VAR
	_bComplete: BOOL; // True if the routing finishes
	_intRet: INT; // Return string converted to an integer
	_bResult : BOOL; // Output of the method
END_VAR
_bResult := FALSE;
bMGetLaserActivatedStatusBusy := TRUE;
_inst_intStep := intMGetLaserActivatedStatusStep;
CASE _inst_intStep OF
	0: // Wait for no error and router not busy
		IF NOT THIS^.P_bError AND NOT bRouterBusy THEN
			bRouterBusy := TRUE;
			_inst_intStep := _inst_intStep + 10;
		END_IF
		
	10: // Initialize parameters
		THIS^.M_LogMessage(_strSTART_MSG);
		_inst_fbParams.M_ClearParameters();
		// ADD ANY PARAMETERS HERE
		_inst_fbParams.M_OutputToParameterList(_inst_arrParams);
		_inst_intStep := _inst_intStep + 10;
		
	20: // Route the command
		_bComplete := M_RouterHelper(
			_in_strMethodName := _strCOMMAND_NAME, 
			_in_timeTimeout := _timeCOMMAND_TIMEOUT,
			_inout_arrParams := _inst_arrParams,
			_inout_arrOutputs := _inst_arrOutputs,
			_out_strReturnValue=>_inst_strRet);
		
		// If route completed, move to next step
		IF _bComplete THEN
			_inst_intStep := _inst_intStep + 10;
			bRouterBusy := FALSE;
		ELSIF THIS^.P_bError THEN
			_inst_intStep := 0;
			bRouterBusy := FALSE;
		END_IF
		
	30: // Parse results
		_intRet := STRING_TO_INT(_inst_strRet);
		IF _intRet > 0 THEN
			_bResult := TRUE;
			THIS^.M_LogMessage(_strEND_MSG);
			// DO ANY PARSING HERE
			_inst_fbParams.M_LoadFromParameterList(_inst_arrOutputs);
			out_IsLaserActivated := _inst_fbParams.M_ParseBool(_inst_fbParams.M_GetParameter('out_IsLaserActivated'));
			bConnected := TRUE;
		// Set error if command failed
		ELSE
			THIS^.M_SetError(_udintERROR_ID, _strERROR_MSG);
		END_IF
		// Go back to start
		_inst_intStep := 0;
END_CASE
M_GetLaserActivatedStatus := _bResult;
intMGetLaserActivatedStatusStep := _inst_intStep;
END_METHOD

METHOD PUBLIC M_GetLaserErrorStatus : BOOL
VAR_INPUT
//	LaserProgramFolderPath : STRING;
END_VAR
VAR_OUTPUT
	out_bool_IsLaserError : BOOL;
END_VAR
VAR CONSTANT
	_strCOMMAND_NAME : T_MaxString	:= 'GetLaserErrorStatus'; // Name of the API method
	_timeCOMMAND_TIMEOUT : TIME		:= T#30S; // Max time to receive API response
	_strSTART_MSG : T_MaxString		:= 'GettingLaserErrorStatus'; // Prints when method starts
	_strEND_MSG : T_MaxString		:= 'ReceivedLaserErrorStatus'; // Prints when method finishes
	_udintERROR_ID : UDINT			:= KeyenceLaserMarkerMDX2000_Error.FailedToGetLaserErrorStatus; // Error ID to set if command fails
	_strERROR_MSG : T_MaxString		:= 'Failed to Get Laser Error Status from Laser Marker!'; // Error message to set if command fails
END_VAR

VAR_INST
	_inst_arrParams: T_ApiParameterList; // Parameters array
	_inst_arrOutputs: T_ApiParameterList; // Outputs array
	_inst_strRet: T_ApiParamValue; // Return string from the router
	_inst_intStep: INT; // Current method step
	_inst_fbParams: FB_ApiParamBuilder; // Parameter builder FB
END_VAR

VAR
	_bComplete: BOOL; // True if the routing finishes
	_intRet: INT; // Return string converted to an integer
	_bResult : BOOL; // Output of the method
END_VAR
_bResult := FALSE;
bMGetLaserErrorStatusBusy := TRUE;
_inst_intStep := intMGetLaserErrorStatusStep;
CASE _inst_intStep OF
	0: // Wait for no error and router not busy
		IF NOT THIS^.P_bError AND NOT bRouterBusy THEN
			bRouterBusy := TRUE;
			_inst_intStep := _inst_intStep + 10;
		END_IF
		
	10: // Initialize parameters
		THIS^.M_LogMessage(_strSTART_MSG);
		_inst_fbParams.M_ClearParameters();
		// ADD ANY PARAMETERS HERE
		_inst_fbParams.M_OutputToParameterList(_inst_arrParams);
		_inst_intStep := _inst_intStep + 10;
		
	20: // Route the command
		_bComplete := M_RouterHelper(
			_in_strMethodName := _strCOMMAND_NAME, 
			_in_timeTimeout := _timeCOMMAND_TIMEOUT,
			_inout_arrParams := _inst_arrParams,
			_inout_arrOutputs := _inst_arrOutputs,
			_out_strReturnValue=>_inst_strRet);
		
		// If route completed, move to next step
		IF _bComplete THEN
			_inst_intStep := _inst_intStep + 10;
			bRouterBusy := FALSE;
		ELSIF THIS^.P_bError THEN
			_inst_intStep := 0;
			bRouterBusy := FALSE;
		END_IF
		
	30: // Parse results
		_intRet := STRING_TO_INT(_inst_strRet);
		IF _intRet > 0 THEN
			_bResult := TRUE;
			THIS^.M_LogMessage(_strEND_MSG);
			// DO ANY PARSING HERE
			_inst_fbParams.M_LoadFromParameterList(_inst_arrOutputs);
			out_bool_IsLaserError := _inst_fbParams.M_ParseBool(_inst_fbParams.M_GetParameter('out_bool_IsLaserError'));
			bConnected := TRUE;
		// Set error if command failed
		ELSE
			THIS^.M_SetError(_udintERROR_ID, _strERROR_MSG);
		END_IF
		// Go back to start
		_inst_intStep := 0;
END_CASE
M_GetLaserErrorStatus := _bResult;
intMGetLaserErrorStatusStep := _inst_intStep;
END_METHOD

METHOD PUBLIC M_GetLaserMarkingStatus : BOOL
VAR_INPUT

END_VAR
VAR_OUTPUT
	out_bool_IsLaserMarking : BOOL;
END_VAR
VAR CONSTANT
	_strCOMMAND_NAME : T_MaxString	:= 'GetLaserMarkingStatus'; // Name of the API method
	_timeCOMMAND_TIMEOUT : TIME		:= T#30S; // Max time to receive API response
	_strSTART_MSG : T_MaxString		:= 'GettingLaserMarkingStatus'; // Prints when method starts
	_strEND_MSG : T_MaxString		:= 'ReceivedLaserMarkingStatus'; // Prints when method finishes
	_udintERROR_ID : UDINT			:= KeyenceLaserMarkerMDX2000_Error.FailedToGetLaserMarkingStatus; // Error ID to set if command fails
	_strERROR_MSG : T_MaxString		:= 'Failed to Get Laser Marking Status from Laser Marker!'; // Error message to set if command fails
END_VAR

VAR_INST
	_inst_arrParams: T_ApiParameterList; // Parameters array
	_inst_arrOutputs: T_ApiParameterList; // Outputs array
	_inst_strRet: T_ApiParamValue; // Return string from the router
	_inst_intStep: INT; // Current method step
	_inst_fbParams: FB_ApiParamBuilder; // Parameter builder FB
END_VAR

VAR
	_bComplete: BOOL; // True if the routing finishes
	_intRet: INT; // Return string converted to an integer
	_bResult : BOOL; // Output of the method
END_VAR
_bResult := FALSE;
bMGetLaserMarkingStatusBusy := TRUE;
_inst_intStep := intMGetLaserMarkingStatusStep;
CASE _inst_intStep OF
	0: // Wait for no error and router not busy
		IF NOT THIS^.P_bError AND NOT bRouterBusy THEN
			bRouterBusy := TRUE;
			_inst_intStep := _inst_intStep + 10;
		END_IF
		
	10: // Initialize parameters
		THIS^.M_LogMessage(_strSTART_MSG);
		_inst_fbParams.M_ClearParameters();
		// ADD ANY PARAMETERS HERE
		_inst_fbParams.M_OutputToParameterList(_inst_arrParams);
		_inst_intStep := _inst_intStep + 10;
		
	20: // Route the command
		_bComplete := M_RouterHelper(
			_in_strMethodName := _strCOMMAND_NAME, 
			_in_timeTimeout := _timeCOMMAND_TIMEOUT,
			_inout_arrParams := _inst_arrParams,
			_inout_arrOutputs := _inst_arrOutputs,
			_out_strReturnValue=>_inst_strRet);
		
		// If route completed, move to next step
		IF _bComplete THEN
			_inst_intStep := _inst_intStep + 10;
			bRouterBusy := FALSE;
		ELSIF THIS^.P_bError THEN
			_inst_intStep := 0;
			bRouterBusy := FALSE;
		END_IF
		
	30: // Parse results
		_intRet := STRING_TO_INT(_inst_strRet);
		IF _intRet > 0 THEN
			_bResult := TRUE;
			THIS^.M_LogMessage(_strEND_MSG);
			// DO ANY PARSING HERE
			_inst_fbParams.M_LoadFromParameterList(_inst_arrOutputs);
			out_bool_IsLaserMarking := _inst_fbParams.M_ParseBool(_inst_fbParams.M_GetParameter('out_bool_IsLaserMarking'));
			bConnected := TRUE;
		// Set error if command failed
		ELSE
			THIS^.M_SetError(_udintERROR_ID, _strERROR_MSG);
		END_IF
		// Go back to start
		_inst_intStep := 0;
END_CASE
M_GetLaserMarkingStatus := _bResult;
intMGetLaserMarkingStatusStep := _inst_intStep;
END_METHOD

METHOD PUBLIC M_GetLaserStatus : BOOL
VAR_INPUT

END_VAR
VAR_OUTPUT
	out_string_laserStatus : STRING;
END_VAR
VAR CONSTANT
	_strCOMMAND_NAME : T_MaxString	:= 'GetLaserStatus'; // Name of the API method
	_timeCOMMAND_TIMEOUT : TIME		:= T#30S; // Max time to receive API response
	_strSTART_MSG : T_MaxString		:= 'GettingLaserStatus'; // Prints when method starts
	_strEND_MSG : T_MaxString		:= 'GotLaserStatus'; // Prints when method finishes
	_udintERROR_ID : UDINT			:= KeyenceLaserMarkerMDX2000_Error.FailedToGetLaserStatus; // Error ID to set if command fails
	_strERROR_MSG : T_MaxString		:= 'Failed to Get Laser Status from Laser Marker!'; // Error message to set if command fails
END_VAR

VAR_INST
	_inst_arrParams: T_ApiParameterList; // Parameters array
	_inst_arrOutputs: T_ApiParameterList; // Outputs array
	_inst_strRet: T_ApiParamValue; // Return string from the router
	_inst_intStep: INT; // Current method step
	_inst_fbParams: FB_ApiParamBuilder; // Parameter builder FB
END_VAR

VAR
	_bComplete: BOOL; // True if the routing finishes
	_intRet: INT; // Return string converted to an integer
	_bResult : BOOL; // Output of the method
END_VAR
_bResult := FALSE;
bMGetLaserStatusBusy := TRUE;
_inst_intStep := intMGetLaserStatusStep;
CASE _inst_intStep OF
	0: // Wait for no error and router not busy
		IF NOT THIS^.P_bError AND NOT bRouterBusy THEN
			bRouterBusy := TRUE;
			_inst_intStep := _inst_intStep + 10;
		END_IF
		
	10: // Initialize parameters
		THIS^.M_LogMessage(_strSTART_MSG);
		_inst_fbParams.M_ClearParameters();
		// ADD ANY PARAMETERS HERE
		_inst_fbParams.M_OutputToParameterList(_inst_arrParams);
		_inst_intStep := _inst_intStep + 10;
		
	20: // Route the command
		_bComplete := M_RouterHelper(
			_in_strMethodName := _strCOMMAND_NAME, 
			_in_timeTimeout := _timeCOMMAND_TIMEOUT,
			_inout_arrParams := _inst_arrParams,
			_inout_arrOutputs := _inst_arrOutputs,
			_out_strReturnValue=>_inst_strRet);
		
		// If route completed, move to next step
		IF _bComplete THEN
			_inst_intStep := _inst_intStep + 10;
			bRouterBusy := FALSE;
		ELSIF THIS^.P_bError THEN
			_inst_intStep := 0;
			bRouterBusy := FALSE;
		END_IF
		
	30: // Parse results
		_intRet := STRING_TO_INT(_inst_strRet);
		IF _intRet > 0 THEN
			_bResult := TRUE;
			THIS^.M_LogMessage(_strEND_MSG);
			// DO ANY PARSING HERE
			_inst_fbParams.M_LoadFromParameterList(_inst_arrOutputs);
			out_string_laserStatus := _inst_fbParams.M_ParseString(_inst_fbParams.M_GetParameter('_out_string_laserStatus'));
			bConnected := TRUE;
		// Set error if command failed
		ELSE
			THIS^.M_SetError(_udintERROR_ID, _strERROR_MSG);
		END_IF
		// Go back to start
		_inst_intStep := 0;
END_CASE
M_GetLaserStatus := _bResult;
intMGetLaserStatusStep := _inst_intStep;
END_METHOD

(* This should clear any errors on the device and bring it to a state where
	it is ready to be energized or otherwise activated. *)
METHOD M_Reset : BOOL
VAR CONSTANT
	_strCOMMAND_NAME : T_MaxString	:= 'Reset'; // Name of the API method
	_timeCOMMAND_TIMEOUT : TIME		:= T#30S; // Max time to receive API response
	_strSTART_MSG : T_MaxString		:= 'Resetting'; // Prints when method starts
	_strEND_MSG : T_MaxString		:= 'Reset'; // Prints when method finishes
	_udintERROR_ID : UDINT			:= KeyenceLaserMarkerMDX2000_Error.FailedToReset; // Error ID to set if command fails
	_strERROR_MSG : T_MaxString		:= 'Failed to reset laser!'; // Error message to set if command fails
	_udintAPI_ERR_ID : UDINT		:= KeyenceLaserMarkerMDX2000_Error.CommandRouterError; // Error to set if there is an error on the API block
	_strAPI_ERR_MSG : T_MaxString	:= 'Error while trying to get API connect status!'; // Error message to set if there is an error on the API block
END_VAR
VAR_INST
	_inst_arrParams: T_ApiParameterList; // Parameters array
	_inst_arrOutputs: T_ApiParameterList; // Outputs array
	_inst_strRet: T_ApiParamValue; // Return string from the router
	_inst_intStep: INT; // Current step
	_inst_fbParams: FB_ApiParamBuilder; // Parameter builder FB
END_VAR
VAR
	_intRet: INT; // Return string converted to an integer
	_bComplete: BOOL; // True if the routing finishes
	_bGotStatus: BOOL; // Goes true once connect status is received
	_bApiConnected: BOOL; // True if API is connected
	_bResult : BOOL; // Output of the method
END_VAR
_bResult := FALSE;
bMResetBusy := TRUE;
_inst_intStep := intMResetStep;
CASE _inst_intStep OF
	0: // Clear errors
		THIS^.M_ClearError();
		in_fbApi.M_ClearError();
		bResetBusy := TRUE;
		_inst_intStep := _inst_intStep + 10;
		
	10: // Check connection status
		_bGotStatus := in_fbApi.M_GetConnectStatus(bConnected => _bApiConnected);
		IF _bGotStatus THEN
			// If the API is connected, go to the next step
			IF _bApiConnected THEN
				_inst_intStep := _inst_intStep + 10;
			// If the API is not connected, reset is done
			ELSE
				_inst_intStep := 0;
				M_Reset := TRUE;
				THIS^.M_LogMessage(_strEND_MSG);
			END_IF
			
		// Set an error 
		ELSIF in_fbApi.P_bError THEN
			_inst_intStep := 0;
			THIS^.M_SetError(_udintAPI_ERR_ID, _strAPI_ERR_MSG);
		END_IF
		
	20: // Wait for router to be free
		IF NOT bRouterBusy THEN
			_inst_intStep := _inst_intStep + 10;
			bRouterBusy := TRUE;
		END_IF
		
	30: // Setup parameters for reset command
		THIS^.M_LogMessage(_strSTART_MSG);
		_inst_fbParams.M_ClearParameters();
		_inst_fbParams.M_OutputToParameterList(_inst_arrParams);
		_inst_intStep := _inst_intStep + 10;
		
	40: // Route command
		_bComplete := M_RouterHelper(
			_in_strMethodName := _strCOMMAND_NAME, 
			_in_timeTimeout := _timeCOMMAND_TIMEOUT,
			_inout_arrParams := _inst_arrParams,
			_inout_arrOutputs := _inst_arrOutputs,
			_out_strReturnValue=>_inst_strRet);
		
		// If route completed, parse results
		IF _bComplete THEN
			_inst_intStep := _inst_intStep + 10;
			bRouterBusy := FALSE;
		ELSIF THIS^.P_bError THEN
			_inst_intStep := 0;
			bRouterBusy := FALSE;
			bResetBusy := FALSE;
		END_IF
		
	50: // Parse results

		// If return value is greater than 1 then robot was reset
		_intRet := STRING_TO_INT(_inst_strRet);
		IF _intRet > 0 THEN
			_bResult := TRUE;
			THIS^.M_LogMessage(_strEND_MSG);
			
		// Else robot failed to reset
		ELSE
			THIS^.M_SetError(_udintERROR_ID, _strERROR_MSG);
		END_IF
		
		// Back to start
		_inst_intStep := 0;
		bResetBusy := FALSE;
END_CASE
M_Reset := _bResult;
intMResetStep := _inst_intStep;
END_METHOD

(* This property should be TRUE while any method in this interface is actively
	executing, or FALSE otherwise. *)
PROPERTY P_bResetBusy : BOOL
GET
END_GET
END_PROPERTY

ACTION A_CommandRecovery:
IF NOT bRouterHelperBusy AND intRouterHelperStep > 0 THEN
	intRouterHelperStep := 0;
	THIS^.M_LogWarning('Router helper ended prematurely!');
END_IF
bRouterHelperBusy := FALSE;

IF NOT bMConnectBusy AND intMConnectStep > 0 THEN
	bRouterBusy := FALSE;
	intMConnectStep := 0;
	THIS^.M_LogWarning('Connect ended prematurely!');
END_IF
bMConnectBusy := FALSE;

IF NOT bMDisconnectBusy AND intMDisconnectStep > 0 THEN
	bRouterBusy := FALSE;
	intMDisconnectStep := 0;
	THIS^.M_LogWarning('Disconnect ended prematurely!');
END_IF
bMDisconnectBusy := FALSE;

IF NOT bMGetConnectStatusBusy AND intMGetConnectStatusStep > 0 THEN
	bRouterBusy := FALSE;
	intMGetConnectStatusStep := 0;
	THIS^.M_LogWarning('Get Connect Status ended prematurely!');
END_IF
bMGetConnectStatusBusy := FALSE;

IF NOT bMPeakCurrentProgramBusy AND intMPeakCurrentProgramStep > 0 THEN
	bRouterBusy := FALSE;
	intMPeakCurrentProgramStep := 0;
	THIS^.M_LogWarning('Peak Current Program ended prematurely!');
END_IF
bMPeakCurrentProgramBusy := FALSE;

IF NOT bMSendMarkingParamsBusy AND intMSendMarkingParamsStep > 0 THEN
	bRouterBusy := FALSE;
	intMSendMarkingParamsStep := 0;
	THIS^.M_LogWarning('Send Marking Params ended prematurely!');
END_IF
bMSendMarkingParamsBusy := FALSE;

IF NOT bMStartMarkingBusy AND intMStartMarkingStep > 0 THEN
	bRouterBusy := FALSE;
	intMStartMarkingStep := 0;
	THIS^.M_LogWarning('Start Marking ended prematurely!');
END_IF
bMStartMarkingBusy := FALSE;

IF NOT bMStopMarkingBusy AND intMStopMarkingStep > 0 THEN
	bRouterBusy := FALSE;
	intMStopMarkingStep := 0;
	THIS^.M_LogWarning('Stop Marking ended prematurely!');
END_IF
bMStopMarkingBusy := FALSE;

IF NOT bMUpdateAllMarkingInfoBusy AND intMUpdateAllMarkingInfoStep > 0 THEN
	bRouterBusy := FALSE;
	intMUpdateAllMarkingInfoStep := 0;
	THIS^.M_LogWarning('Update All Marking Info ended prematurely!');
END_IF
bMUpdateAllMarkingInfoBusy := FALSE;

IF NOT bMUpdateSingleBlockInfoBusy AND intMUpdateSingleBlockInfoStep > 0 THEN
	bRouterBusy := FALSE;
	intMUpdateSingleBlockInfoStep := 0;
	THIS^.M_LogWarning('Update Single Block Info ended prematurely!');
END_IF
bMUpdateSingleBlockInfoBusy := FALSE;

IF NOT bMGetCurrentProgBusy AND intMGetCurrentProgStep > 0 THEN
	bRouterBusy := FALSE;
	intMGetCurrentProgStep := 0;
	THIS^.M_LogWarning('Get Current Program ended prematurely!');
END_IF
bMGetCurrentProgBusy := FALSE;

IF NOT bMLoadProgramBusy AND intMLoadProgramStep > 0 THEN
	bRouterBusy := FALSE;
	intMLoadProgramStep := 0;
	THIS^.M_LogWarning('Load Program ended prematurely!');
END_IF
bMLoadProgramBusy := FALSE;

IF NOT bMSaveCurrentLaserProgramtoPCBusy AND intMSaveCurrentLaserProgramtoPC > 0 THEN
	bRouterBusy := FALSE;
	intMSaveCurrentLaserProgramtoPC := 0;
	THIS^.M_LogWarning('Save Current Laser Program to PC ended prematurely!');
END_IF
bMSaveCurrentLaserProgramtoPCBusy := FALSE;

IF NOT bMSendProgramToLaserBusy AND intMSendProgramToLaserStep > 0 THEN
	bRouterBusy := FALSE;
	intMSendProgramToLaserStep := 0;
	THIS^.M_LogWarning('Send Program to Laser ended prematurely!');
END_IF
bMSendProgramToLaserBusy := FALSE;

IF NOT bMStartProgramBusy AND intMStartProgramStep > 0 THEN
	bRouterBusy := FALSE;
	intMStartProgramStep := 0;
	THIS^.M_LogWarning('Start Program ended prematurely!');
END_IF
bMStartProgramBusy := FALSE;

IF NOT bMUpdateSingleProgramBlockDataBusy AND intMUpdateSingleProgramBlockDataStep > 0 THEN
	bRouterBusy := FALSE;
	intMUpdateSingleProgramBlockDataStep := 0;
	THIS^.M_LogWarning('Update Single Program Block Data ended prematurely!');
END_IF
bMUpdateSingleProgramBlockDataBusy := FALSE;

IF NOT bMUpdateSingleProgramBlockMarkingEnabledBusy AND intMUpdateSingleProgramBlockMarkingEnabledStep > 0 THEN
	bRouterBusy := FALSE;
	intMUpdateSingleProgramBlockMarkingEnabledStep := 0;
	THIS^.M_LogWarning('Update Single Program Block Marking Enabled ended prematurely!');
END_IF
bMUpdateSingleProgramBlockMarkingEnabledBusy := FALSE;

IF NOT bMGetLaserActivatedStatusBusy AND intMGetLaserActivatedStatusStep > 0 THEN
	bRouterBusy := FALSE;
	intMGetLaserActivatedStatusStep := 0;
	THIS^.M_LogWarning('Get Laser Activated Status ended prematurely!');
END_IF
bMGetLaserActivatedStatusBusy := FALSE;

IF NOT bMGetLaserErrorStatusBusy AND intMGetLaserErrorStatusStep > 0 THEN
	bRouterBusy := FALSE;
	intMGetLaserErrorStatusStep := 0;
	THIS^.M_LogWarning('Get Laser Error Status ended prematurely!');
END_IF
bMGetLaserErrorStatusBusy := FALSE;

IF NOT bMGetLaserMarkingStatusBusy AND intMGetLaserMarkingStatusStep > 0 THEN
	bRouterBusy := FALSE;
	intMGetLaserMarkingStatusStep := 0;
	THIS^.M_LogWarning('Get Laser Marking Status ended prematurely!');
END_IF
bMGetLaserMarkingStatusBusy := FALSE;

IF NOT bMGetLaserStatusBusy AND intMGetLaserStatusStep > 0 THEN
	bRouterBusy := FALSE;
	intMGetLaserStatusStep := 0;
	THIS^.M_LogWarning('Get Laser Status ended prematurely!');
END_IF
bMGetLaserStatusBusy := FALSE;

IF NOT bMClearErrorBusy AND intMClearErrorStep > 0 THEN
	bRouterBusy := FALSE;
	intMClearErrorStep := 0;
	THIS^.M_LogWarning('Clear Error ended prematurely!');
END_IF
bMClearErrorBusy := FALSE;

IF NOT bMResetBusy AND intMResetStep > 0 THEN
	bRouterBusy := FALSE;
	intMResetStep := 0;
	THIS^.M_LogWarning('Reset ended prematurely!');
END_IF
bMResetBusy := FALSE;
END_ACTION

(*
Sends the given method to the API and receives and partially parses the result.
*)
METHOD PRIVATE M_RouterHelper : BOOL
VAR_INPUT
	(* Name of the method to call. *)
	_in_strMethodName : T_MaxString;
	(* Maximum time to wait for method response. *)
	_in_timeTimeout : TIME;
END_VAR
VAR_IN_OUT
	(* The array of parameters to send to the API. *)
	_inout_arrParams : T_ApiParameterList;
	(* The array that gets populated with any method output data. *)
	_inout_arrOutputs : T_ApiParameterList;
END_VAR
VAR_OUTPUT
	(* JSON string of the method return value. *)
	_out_strReturnValue: T_ApiParamValue;
END_VAR
VAR_INST
	(* Current step. *)
	_inst_intStep: INT;
	(* True if the method executed. *)
	_inst_bExec: BOOL;
	(* Return string of the method. *)
	_inst_strRet: T_ApiParamValue;
END_VAR
VAR
	(* True once the command routing finishes. *)
	_bComplete: BOOL;
	(* True once the API connects. *)
	_bApiConnect: BOOL;
END_VAR
bRouterHelperBusy := TRUE;
_inst_intStep := intRouterHelperStep;
CASE _inst_intStep OF
	0: // Start process only if there is no error on this FB
		IF NOT THIS^.P_bError THEN
			in_fbApi.M_ClearError();
			_inst_intStep := 10;
		END_IF
		
	10: // Check if command router connected
		IF NOT in_fbApi.P_bConnected THEN
			_inst_intStep := 20; // Go to API connect step
		ELSE
			_inst_intStep := 30; // Go to route command step
		END_IF
		
	20: // Connect the command router
		_bApiConnect := in_fbApi.M_Connect();
		IF _bApiConnect THEN
			_inst_intStep := _inst_intStep + 10; // Go to next step
		ELSIF in_fbApi.P_bError THEN
			THIS^.M_SetError(KeyenceLaserMarkerMDX2000_Error.CommandRouterError, 'Error on command router function block while connecting!');
			_inst_intStep := 0; // Go back to start
		END_IF
		
	30:	// Route the command
		_bComplete := in_fbApi.M_RouteCommand(
			_in_strModuleId := in_strUniqueId,
			_in_strMethodName := _in_strMethodName,
			_in_timeTimeout := _in_timeTimeout,
			_inout_arrParameters := _inout_arrParams,
			_inout_arrOutputs := _inout_arrOutputs,
			_out_bCommandExecuted => _inst_bExec,
			_out_strReturnValue => _inst_strRet);
		IF _bComplete THEN
			_inst_intStep := _inst_intStep + 10; // Go to next step
		ELSIF in_fbApi.P_bError THEN
			THIS^.M_SetError(KeyenceLaserMarkerMDX2000_Error.CommandRouterError, 'Error on command router function block while routing command!');
			_inst_intStep := 0; // Go back to start
		END_IF
		
	40: // Check result then go back to start
		IF NOT _inst_bExec THEN
			THIS^.M_SetError(KeyenceLaserMarkerMDX2000_Error.CommandFault, 'Method in API failed to execute!');
		ELSE
			_out_strReturnValue := _inst_strRet;
			M_RouterHelper := TRUE;
		END_IF
		_inst_intStep := 0; // Go back to start
END_CASE
intRouterHelperStep := _inst_intStep;
END_METHOD

END_FUNCTION_BLOCK

// Project Information/F_GetCompany
// This function has been automatically generated from the project information.
{attribute 'signature_flag' := '1073741824'}
{attribute 'TcGenerated'}
{attribute 'no-analysis'}
FUNCTION F_GetCompany : WSTRING
VAR_INPUT
	
END_VAR

F_GetCompany := "Sensata Technologies";

END_FUNCTION

// Project Information/F_GetTitle
// This function has been automatically generated from the project information.
{attribute 'signature_flag' := '1073741824'}
{attribute 'TcGenerated'}
{attribute 'no-analysis'}
FUNCTION F_GetTitle : WSTRING
VAR_INPUT
	
END_VAR

F_GetTitle := "Sensata_Laser";

END_FUNCTION

// Project Information/F_GetVersion
// This function has been automatically generated from the project information.
{attribute 'signature_flag' := '1073741824'}
{attribute 'TcGenerated'}
{attribute 'no-analysis'}
FUNCTION F_GetVersion : ST_LibVersion
VAR_INPUT
	
END_VAR

F_GetVersion.iMajor := 1;
F_GetVersion.iMinor := 0;
F_GetVersion.iBuild := 1;
F_GetVersion.iRevision := 0;
F_GetVersion.sVersion := '1.0.1';
F_GetVersion.nFlags := 0;

END_FUNCTION
